// TwinCAT 3 PLC project Untitled1
// ProgramVersion: 3.1.4023.0
// libraries:
//   Tc2_Standard, * (Beckhoff Automation GmbH)
//   Tc2_System, * (Beckhoff Automation GmbH)
//   Tc2_Utilities, * (Beckhoff Automation GmbH)
//   Tc3_Module, * (Beckhoff Automation GmbH)
//   VisuSymbols,3.5.10.0,System
// project tree:
//   / GlobalTextList.TcGTLO, PlcTask.TcTTO, Visualization Manager.TcVMO (not stored)
//   GVLs/ GVL.TcGVL
//   POUs/ MAIN.TcPOU
//   VISUs/ Visualization.TcVIS
// real-time tasks:
//   TASK PlcTask: cycle T#10ms, priority 20, ADS port 350
// I/O:
//   DEVICE Device 2 (EtherCAT), AmsNetId 10.40.1.85.3.1
//     Term 1 (EK1100) [EK1100 EtherCAT Coupler (2A E-Bus)]
//       Term 6 (EL7041) [EL7041 1Ch. Stepper motor output stage (50V, 5A)]
//       Term 3 (EL1809) [EL1809 16Ch. Dig. Input 24V, 3ms]
//       Term 5 (EL9011) [EL9011 End Terminal]
//     Box 4 (EasyCAT 32+32 rev 1) [Generic 32+32 bytes rev 1]
// variable links:
//   Untitled1/Untitled1 Instance <-> Device 2 (EtherCAT)/Box 4 (EasyCAT 32+32 rev 1)
//     PlcTask Inputs/MAIN.Analog1 <-> Inputs/Byte0
//     PlcTask Inputs/MAIN.Analog2 <-> Inputs/Byte1
//     PlcTask Inputs/MAIN.Analog3 <-> Inputs/Byte2
//     PlcTask Inputs/MAIN.Analog4 <-> Inputs/Byte4
//     PlcTask Inputs/MAIN.Analog5 <-> Inputs/Byte5
//     PlcTask Inputs/MAIN.Analog6 <-> Inputs/Byte6
//     PlcTask Inputs/MAIN.Analog7 <-> Inputs/Byte8
//     PlcTask Inputs/MAIN.Analog8 <-> Inputs/Byte9
//     PlcTask Inputs/MAIN.Analog9 <-> Inputs/Byte10
//     PlcTask Inputs/MAIN.Average <-> Inputs/Byte3
//     PlcTask Inputs/MAIN.AverageLeft <-> Inputs/Byte7
//     PlcTask Inputs/MAIN.AverageRight <-> Inputs/Byte11
//     PlcTask Inputs/MAIN.Byte31IN <-> Inputs/Byte31
//     PlcTask Inputs/MAIN.Sensors <-> Inputs/Byte12
//     PlcTask Outputs/GVL.ArduinoState <-> Outputs/Byte0
//     PlcTask Outputs/GVL.FanDyno <-> Outputs/Byte1
//     PlcTask Outputs/GVL.OutArduino <-> Outputs/Byte2
//   Untitled1/Untitled1 Instance <-> Device 2 (EtherCAT)/Term 1 (EK1100)/Term 6 (EL7041)
//     PlcTask Inputs/GVL.CounterVal <-> ENC Status/Counter value
//     PlcTask Outputs/GVL.EnableMotor <-> STM Control/Control/Enable
//     PlcTask Outputs/GVL.ReduceTorqueMotor <-> STM Control/Control/Reduce torque
//     PlcTask Outputs/GVL.ResetMotor <-> STM Control/Control/Reset
//     PlcTask Outputs/GVL.SetCounter <-> ENC Control/Control/Set counter
//     PlcTask Outputs/GVL.SetCounterVal <-> ENC Control/Set counter value
//     PlcTask Outputs/GVL.VelocityMotor <-> STM Velocity/Velocity

CONFIGURATION Untitled1
    RESOURCE PLC ON TwinCAT3
        TASK PlcTask(INTERVAL := T#10ms, PRIORITY := 20);
        PROGRAM MAIN WITH PlcTask : MAIN;
    END_RESOURCE
END_CONFIGURATION

// ---- GVLs/GVL.TcGVL
{attribute 'qualified_only'}
VAR_GLOBAL
	SystemTime							:WORD;
	SystemTimeM							:WORD;
	SystemTimeMs						:WORD;
	LeftAirJet							:BOOL;
	RightAirJet							:BOOL;
	AirJet1								:BOOL;
	AirJet2								:BOOL;
	ArduinoState 				AT %Q*	:USINT		:=0;//byte out 0
	OutArduino					AT %Q*	:USINT;//byte out 2
	FanDyno						AT %Q*	:USINT		:=0; //byte out 1
	CounterVal					AT %I*	:UDINT;
	SetCounter					AT %Q*	:BOOL;
	SetCounterVal				AT %Q*	:UDINT;
	EnableMotor					AT %Q*	:BOOL;//stm enable
	ResetMotor					AT %Q*	:BOOL;
	ReduceTorqueMotor			AT %Q*	:BOOL;
	ExecutePosMotor				AT %Q*	:BOOL;
	EmergencyStopMotor			AT %Q*	:BOOL;
	TargetPosMotor				AT %Q*	:UDINT;
	VelocityMotor 				AT %Q*	:INT;
	AccelMotor 					AT %Q*	:INT := 150;
	DecelMotor 					AT %Q*	:INT :=150;
	StartTypeMotor				AT %Q*	:UINT;
	MotorPos					AT %I*	:UDINT;
	StepperUp							:BOOL;
	StepperDown							:BOOL;
END_VAR

// ---- POUs/MAIN.TcPOU
PROGRAM MAIN
VAR
	Analog1   		AT %I*	:USINT;//byte in 0
	Analog2   		AT %I*	:USINT;//byte in 1
	Analog3   		AT %I*	:USINT;//byte in 2
	Average   		AT %I*	:USINT;//byte in 3
	Analog4   		AT %I*	:USINT;//byte in 4
	Analog5   		AT %I*	:USINT;//byte in 5
	Analog6   		AT %I*	:USINT;//byte in 6
	AverageLeft  	AT %I*	:USINT;//byte in 7
	Analog7   		AT %I*	:USINT;//byte in 8  CLOSE WING
	Analog8   		AT %I*	:USINT;//byte in 9  CLOSE WING
	Analog9   		AT %I*	:USINT;//byte in 10 CLOSE WING
	AverageRight   	AT %I*	:USINT;//byte in 11 CLOSE WING
	Sensors			AT %I*	:USINT;//byte in 12

	Number					:INT;
	Scanner					:USINT		:= 10;
	Idle					:USINT		:= 0;
	WingGo					:USINT		:=20;
	FanGo					:USINT		:=30;
	PlixFanGo				:USINT		:=40;
	State					:INT 		:=0;

	Byte31IN		AT %I*	:USINT;
	ArduinoBusyBit			:BOOL;
	ArduinoComsTimer		:TON;
	EndStopTimer			:TON;
	StackSensor1			:BOOL;
	StackSensor2			:BOOL;
	StackSensor3			:BOOL;
	TopEndStop		AT %I*	:BOOL;
	BottomEndStop	AT %I*	:BOOL;
	
	AirJet3					:BOOL;
	Sensor4					:BOOL;
	Sensor5					:BOOL;
	PlixNumber				:INT;
	Delay 					:TON;
	RampTimer				:TON;
  	Count 					:INT		:= 0;
	e 						:INT;
	Up						:INT		:=850;
	Down					:INT		:=-950;
	fbTime					:FB_LocalSystemTime := ( bEnable :=TRUE, dwCycle := 1 );
	StartTime				:REAL;
	GoTime					:REAL;
	EndTime					:REAL;
	TotalTime				:REAL;
	CycleTime				:REAL;
	AverageTime				:REAL;
	TimeSeconds				:REAL;
	StepperUp				:BOOL;
	StepperDown				:BOOL;
	Singles					:INT;
	Doubles					:INT;
	Single					:BOOL;
	Double					:BOOL;
	Zero					:BOOL;
	Zeros					:INT;
	msgCtrlMask     		:DWORD;
    msgFmtStr               :T_MaxString;
    strArg          		:T_MaxString;
	Calibrate 				:BOOL;
	TopPickScan				:INT;
	HalfWayDownScan			:INT;
	
	
	TopPickCut				:INT;
	HalfWayCut				:INT;
	Wiggle					:INT;
	TopCount				:UDINT;

END_VAR

VAR PERSISTENT
	TopCut					:INT;
	BottomCut				:INT;
	TopCutLeft				:INT;
	BottomCutLeft			:INT;
	TopCutRight				:INT;
	BottomCutRight			:INT;
	PlixNumberScan			:INT;
	PlixNumberScanLeft		:INT;
	PlixNumberScanRight		:INT;
	ArduinoComsTime			:TIME		:=T#10MS;
	EndStopTime				:TIME		:=T#500MS;
	RampTime				:TIME		:=T#500MS;
END_VAR

ArduinoBusyBit := Byte31IN.0;
StackSensor1 := Sensors.0;
StackSensor2 := Sensors.1;
StackSensor3 := Sensors.2;
Sensor4 := Sensors.3;
Sensor5 := Sensors.4;
GVL.OutArduino.0 := GVL.AirJet1;
GVL.OutArduino.1 := GVL.AirJet2;
GVL.OutArduino.2 := AirJet3;
GVL.OutArduino.3 := GVL.LeftAirJet;
GVL.OutArduino.4 := GVL.RightAirJet;

GVL.SystemTime := fbTime.systemTime.wSecond;
GVL.SystemTimeMs := fbTime.systemTime.wMilliseconds;
GVL.SystemTimeM := fbTime.systemTime.wMinute;
TimeSeconds := GVL.SystemTime + (GVL.SystemTimeMs * 0.001) + ( GVL.SystemTimeM * 60 );

ArduinoComsTimer(
	IN := GVL.ArduinoState > 0,
	PT := ArduinoComsTime,);
	
IF ArduinoComsTimer.Q THEN
	GVL.ArduinoState := Idle;
END_IF
	
IF GVL.StepperDown THEN
	IF GVL.VelocityMotor < 2500 THEN
		GVL.VelocityMotor := GVL.VelocityMotor +100;
	ELSE
		GVL.VelocityMotor :=2500;
	END_IF
END_IF

IF GVL.StepperUp THEN
	IF GVL.VelocityMotor > -2500 THEN
		GVL.VelocityMotor := GVL.VelocityMotor -100;
	ELSE
		GVL.VelocityMotor :=-2500;
	END_IF
END_IF
IF (GVL.CounterVal > 5070000) AND (State >2000) THEN//reeundant
	GVL.VelocityMotor :=0;
	GVL.StepperUp := FALSE;
	GVL.StepperDown := FALSE;
END_IF

GVL.EnableMotor := TRUE;
fbTime();


CASE State OF

	100:
		
		IF NOT StackSensor1 THEN//AND NOT StackSensor2 AND NOT StackSensor3 THEN
			GVL.StepperDown := TRUE;
		ELSE 
			GVL.VelocityMotor :=0;
			GVL.StepperUp := FALSE;
			GVL.StepperDown := FALSE;
			State :=200;
			
		END_IF
	
	200:
		
		Delay(IN:=TRUE, PT:=T#100MS);
      	IF Delay.Q THEN
        	Delay(IN:=FALSE);
			State := 300;
		END_IF
	
	300:
		IF StackSensor1 THEN//AND NOT StackSensor2 AND NOT StackSensor3 THEN
			GVL.StepperUp := TRUE;
		ELSE 
			GVL.VelocityMotor :=0;
			GVL.StepperUp := FALSE;
			GVL.StepperDown := FALSE;
			GVL.SetCounterVal :=5000000;
			GVL.SetCounter :=TRUE;
			State :=400;
				
			END_IF
	
	400:
		GVL.SetCounter :=FALSE;
		Delay(IN:=TRUE, PT:=T#200MS);
      	IF Delay.Q THEN
        	Delay(IN:=FALSE);
			State := 500;
			TopCount := GVL.CounterVal - 19000;
		END_IF
		
		
	500:
	IF ArduinoBusyBit THEN//if arduino is free then ask to change state
		GVL.FanDyno :=103;
		GVL.ArduinoState := FanGo;
        State := 600;
	END_IF
	600:
		Delay(IN:=TRUE, PT:=T#200MS);
      	IF Delay.Q THEN
        	Delay(IN:=FALSE);
			State := 700;
		END_IF
	700:
		GVL.ArduinoState := Scanner;
		IF (GVL.CounterVal > TopCount) AND (Average > 200) THEN
			GVL.StepperUp := TRUE;
		ELSE 
			GVL.VelocityMotor :=0;
			GVL.StepperUp := FALSE;
			GVL.StepperDown := FALSE;
			State :=800;
		END_IF		
	800:
		IF (GVL.CounterVal < 5012000) THEN
			GVL.StepperDown := TRUE;
		ELSE 
			GVL.VelocityMotor :=0;
			GVL.StepperUp := FALSE;
			GVL.StepperDown := FALSE;
			State :=900;
		END_IF	

	900:	
		Delay(IN:=TRUE, PT:=T#300MS);
      	IF Delay.Q THEN
        	Delay(IN:=FALSE);
			State := 1000;
		END_IF
	1000:
		IF ArduinoBusyBit THEN
			GVL.ArduinoState := Scanner;
			State := 1100;
		END_IF
		
		
	1100:
		Delay(IN:=TRUE, PT:=T#1000MS);
      	IF Delay.Q THEN
        	Delay(IN:=FALSE);
			State := 1200;
		END_IF
	1200:
		
		IF Average > 200 THEN//repick
			PlixNumber := 0;
			Zeros := Zeros + 1;
			State := 100;
		ELSIF Average >=BottomCut AND Average <TopCut THEN//good
			PlixNumber := 1;
			Single := TRUE;
			State := 2000;
		ELSIF Average >=TopCut THEN//wiggle process
			Double := TRUE;
			State := 1300;
		END_IF
		IF Calibrate THEN
			Single := TRUE;
		 	PlixNumberScan := Average;
			PlixNumberScanLeft :=AverageLeft;
			PlixNumberScanRight :=AverageRight;
			State := 2500;
		END_IF
		
		IF Average < BottomCut THEN//good
			PlixNumber := 2;
			Single := TRUE;
			State := 2000;
		ELSIF Average >=BottomCut AND Average <TopCut THEN//double
			PlixNumber := 2;
			Double := TRUE;
			State := 1300;
		ELSIF Average >=TopCut THEN//repick
			PlixNumber := 0;
			Zeros := Zeros + 1;
			State := 100;
		END_IF
		IF Calibrate THEN
			Single := TRUE;
		 	PlixNumberScan := Average;
			PlixNumberScanLeft :=AverageLeft;
			PlixNumberScanRight :=AverageRight;
			State := 2500;
		END_IF
		
		
	1300:
		IF AverageLeft < TopCut +60 AND AverageRight > TopCut +60 THEN
			GVL.LeftAirJet := TRUE;
			State := 1350;
		ELSIF AverageLeft > TopCut+60 AND AverageRight < TopCut +60  THEN
			GVL.RightAirJet := TRUE;
			State := 1350;
		ELSE 
			State := 1400;
		END_IF
		
	1350:
		Delay(IN:=TRUE, PT:=T#500MS);
		IF Delay.Q THEN
			Delay(IN:=FALSE);
			GVL.LeftAirJet := FALSE;
			GVL.RightAirJet := FALSE;
			State := 1351;
		END_IF
	1351:
		Delay(IN:=TRUE, PT:=T#200MS);
		IF Delay.Q THEN
			Delay(IN:=FALSE);
			State := 1000;
		END_IF
	1400:
		Wiggle := Wiggle +1;
		IF ArduinoBusyBit THEN//if arduino is free then ask to change state
			GVL.FanDyno :=130;
			GVL.ArduinoState := WingGo;
			Delay(IN:=TRUE, PT:=T#500MS);
			IF Delay.Q THEN
				Delay(IN:=FALSE);
				State := 1450; 
			END_IF
		END_IF
	1450:
		IF ArduinoBusyBit THEN//if arduino is free then ask to change state
			GVL.FanDyno :=200;
			GVL.ArduinoState := WingGo;
			Delay(IN:=TRUE, PT:=T#500MS);
			IF Delay.Q THEN
				Delay(IN:=FALSE);
				State := 1500;
			END_IF
		END_IF
	1500:
		GVL.FanDyno :=170;
		GVL.ArduinoState := WingGo;
		Delay(IN:=TRUE, PT:=T#500MS);
		IF Delay.Q THEN
			Delay(IN:=FALSE);
			State := 1000;
		END_IF
	
	
	
	2000:
		//GVL.StepperDown := TRUE;
		State :=2100;
		
	2100:
		GVL.FanDyno := 74;
		GVL.ArduinoState := 30;
		State:=2200;
	2200:
		Delay(IN:=TRUE, PT:=T#100MS);
		IF Delay.Q THEN
        	Delay(IN:=FALSE);
        	State := 2300;
    	END_IF
	2300:
		GVL.AirJet2 :=TRUE;
		State := 2400;
	2400:
		Delay(IN:=TRUE, PT:=T#300MS);
		IF Delay.Q THEN
        	Delay(IN:=FALSE);
        	State := 2500;
    	END_IF
	2500:
		GVL.FanDyno := 89;
		GVL.ArduinoState := 30;
		State := 2600;
	
	2600:
		Delay(IN:=TRUE, PT:=T#100MS);
		IF Delay.Q THEN
        	Delay(IN:=FALSE);
			GVL.AirJet2 :=FALSE;
        	State := 2800;
    	END_IF
	2800:
	//finishing up stats ant time and stuff
		State :=100;
		IF Single THEN
			Singles := Singles +1;
		END_IF
		IF Double THEN
			Doubles := Doubles +1;
		END_IF
		Single := FALSE;
		Double := FALSE;
		EndTime := TimeSeconds;	
		AverageTime := (EndTime - GoTime)/Singles;
		CycleTime := EndTime - StartTime;
		IF Calibrate THEN
			Singles := Singles -1;
			TopCut := Average + 140;
			BottomCut := Average + 40;
			TopCutLeft := AverageLeft - 40;
			BottomCutLeft := AverageLeft - 66;
			TopCutRight := AverageRight + 10;
			BottomCutRight := AverageRight - 50;
			State :=0;
			Calibrate := FALSE;
		END_IF
			
		
	
END_CASE

END_PROGRAM

// ---- GlobalTextList.TcGTLO
TEXTLIST GlobalTextList
  481 = '%d'
  432 = '%f'
  79 = 'Average'
  745 = 'Blast Air'
  656 = 'Calibrate'
  311 = 'Cycle'
  443 = 'DOWN'
  953 = 'Down'
  71 = 'down'
  17 = 'Encoder zero'
  197 = 'Fan'
  407 = 'fan off'
  680 = 'flat'
  214 = 'GO'
  969 = 'Half Down'
  638 = 'High'
  143 = 'Hold'
  189 = 'Left Air'
  752 = 'Left Wing'
  971 = 'Mid'
  628 = 'Motor reset'
  454 = 'Off'
  750 = 'Reverse'
  187 = 'Right Air'
  681 = 'Right Wing'
  757 = 'Scan'
  942 = 'Shoot Air'
  150 = 'Stop'
  468 = 'UP'
  375 = 'up'
  646 = 'WINGS'
  357 = 'Zero stats'
END_TEXTLIST

// ---- VISUs/Visualization.TcVIS
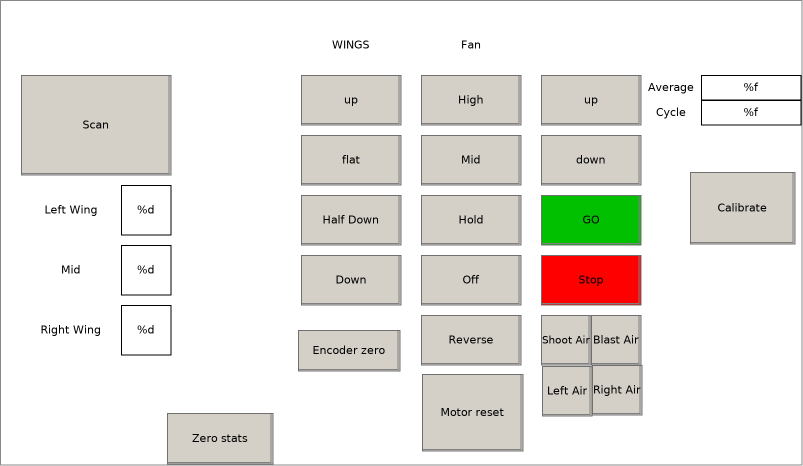
VISUALIZATION Visualization  // 803x466
    Button (422,374 101x77), "Motor reset"
        OnMouseDown: execute { GVL.ResetMotor :=TRUE; }
        OnMouseUp: execute { GVL.ResetMotor :=FALSE; }
    Button (21,75 150x100), "Scan"
        OnMouseDown: execute { GVL.ArduinoState := MAIN.Scanner; }
    Button (301,75 100x50), "up"
        OnMouseDown: execute { GVL.FanDyno :=220 GVL.ArduinoState := MAIN.WingGo }
    Button (301,135 100x50), "flat"
        OnMouseDown: execute { GVL.FanDyno :=180 GVL.ArduinoState := MAIN.WingGo }
    Button (301,255 100x50), "Down"
        OnMouseDown: execute { GVL.FanDyno :=80 GVL.ArduinoState := MAIN.WingGo }
    Button (301,195 100x50), "Half Down"
        OnMouseDown: execute { GVL.FanDyno :=155 GVL.ArduinoState := MAIN.WingGo }
    Label (301,20 100x50), "WINGS"
    Button (421,75 100x50), "High"
        OnMouseDown: execute { GVL.FanDyno :=103 GVL.ArduinoState := MAIN.FanGo }
    Button (421,135 100x50), "Mid"
        OnMouseDown: execute { GVL.FanDyno :=100 GVL.ArduinoState := MAIN.FanGo }
    Button (421,255 100x50), "Off"
        OnMouseDown: execute { GVL.FanDyno :=89 GVL.ArduinoState := MAIN.FanGo }
    Button (421,195 100x50), "Hold"
        OnMouseDown: execute { GVL.FanDyno :=97 GVL.ArduinoState := MAIN.FanGo }
    Label (421,20 100x50), "Fan"
    Button (421,315 100x50), "Reverse"
        OnMouseDown: execute { GVL.FanDyno :=74 GVL.ArduinoState := MAIN.FanGo }
    Button (541,195 100x50), "GO"
        OnMouseUp: execute { MAIN.State := 100; MAIN.GoTime := MAIN.TimeSeconds; }
    Button (541,255 100x50), "Stop"
        OnMouseDown: execute {
            MAIN.State := 0;
            GVL.ArduinoState := 0;
            GVL.StepperUp := FALSE;
            GVL.StepperDown := FALSE;
            GVL.VelocityMotor :=0;
            MAIN.TotalTime := MAIN.TimeSeconds;
        }
    Button (541,315 50x50), "Shoot Air"
        OnMouseDown: execute { GVL.AirJet2 := TRUE; }
        OnMouseUp: execute { GVL.AirJet2 := FALSE; }
    Button (591,315 50x50), "Blast Air"
        OnMouseDown: execute { GVL.AirJet1 := TRUE; }
        OnMouseUp: execute { GVL.AirJet1 := FALSE; }
    Button (541,75 100x50), "up"
        OnMouseDown: execute { GVL.StepperUp	:= TRUE; }
        OnMouseUp: execute { GVL.StepperUp	:= FALSE; GVL.VelocityMotor :=0; }
    Button (541,135 100x50), "down"
        OnMouseDown: execute { GVL.StepperDown	:= TRUE; }
        OnMouseUp: execute { GVL.StepperDown	:= FALSE; GVL.VelocityMotor :=0; }
    Rectangle (701,75 100x25), "%f", text variable: MAIN.AverageTime
    Rectangle (701,100 100x25), "%f", text variable: MAIN.CycleTime
    Label (621,75 100x25), "Average"
    Label (621,100 100x25), "Cycle"
    Button (690,172 105x72), "Calibrate"
        OnMouseDown: execute {
            MAIN.Calibrate := TRUE;
            MAIN.State := 100;
            MAIN.GoTime := MAIN.TimeSeconds;
        }
    Rectangle (121,185 50x50), "%d", text variable: MAIN.AverageLeft
    Rectangle (121,245 50x50), "%d", text variable: MAIN.Average
    Rectangle (121,305 50x50), "%d", text variable: MAIN.AverageRight
    Label (21,185 100x50), "Left Wing"
    Label (21,245 100x50), "Mid"
    Label (21,305 100x50), "Right Wing"
    Button (298,330 102x41), "Encoder zero"
        OnMouseDown: execute { GVL.SetCounterVal :=5000000; GVL.SetCounter :=TRUE; }
        OnMouseUp: execute {
            //ShooterBob.EncoderCount :=FALSE;
        }
    Button (542,366 50x50), "Left Air"
        OnMouseDown: execute { GVL.LeftAirJet := TRUE; }
        OnMouseUp: execute { GVL.LeftAirJet := FALSE; }
    Button (592,365 50x50), "Right Air"
        OnMouseDown: execute { GVL.RightAirJet := TRUE; }
        OnMouseUp: execute { GVL.RightAirJet := FALSE; }
    Button (167,413 106x51), "Zero stats"
        OnMouseDown: execute {
            MAIN.Singles :=0;
            MAIN.Doubles :=0;
            MAIN.Wiggle :=0;
            MAIN.Zeros :=0;
            MAIN.AverageTime :=0;
            MAIN.CycleTime := 0;
            MAIN.GoTime := 0;
            MAIN.EndTime  := 0;
            MAIN.StartTime := 0;
        }
END_VISUALIZATION
